{attribute 'linkalways'} 
{attribute 'no_explicit_call' := 'This FB is a CLASS and must be accessed using methods or properties'}
{attribute 'enable_dynamic_creation'}
FUNCTION_BLOCK ParameterUpdatedEvent EXTENDS Disposable IMPLEMENTS I_ParameterUpdatedEvent
VAR
	_targetParameter : I_Parameter;
END_VAR

METHOD FB_init : BOOL
VAR_INPUT
	bInitRetains : BOOL; // if TRUE, the retain variables are initialized (warm start / cold start)
	bInCopyCode : BOOL;  // if TRUE, the instance afterwards gets moved into the copy code (online change)
	TargetParameter : I_Parameter;
END_VAR
THIS^._targetParameter := TargetParameter;
END_METHOD

PROPERTY PUBLIC TargetParameter : I_Parameter
GET
TargetParameter := _targetParameter;
END_GET
END_PROPERTY

END_FUNCTION_BLOCK

(* stored: Version 1.1.0.1, ProductVersion 3.1.4024.13
   POU ParameterUpdatedEvent: Id {9aee1605-6915-0070-07cf-dca051deefd5}, SpecialFunc None
   Folder Constructor: Id {ea62013f-407f-00ab-2a44-7b880f9ea242}
   Method FB_init: Id {df25cc75-92c3-0f66-2229-5ce0b212a433}
   Property TargetParameter: Id {1a47f78c-f489-0205-0800-4797f8a803e0}
   Get Get: Id {8dd4471b-1a99-0f37-237e-c62371e6869c} *)
